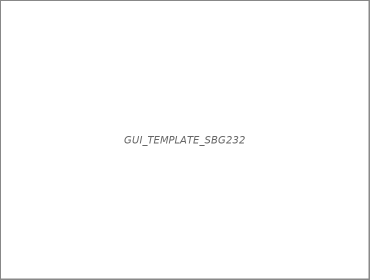
VISUALIZATION GUI_SBG232_SIM  // 370x280
    Frame (0,0 370x280)
        shows GUI_TEMPLATE_SBG232(m_Instance := MAIN.sbg232_sim)
END_VISUALIZATION

(* stored: Version 1.1.0.1, ProductVersion 3.1.4024.12
   Visu GUI_SBG232_SIM: Id {af8018f8-06c7-4b23-aad0-1f1dba0308bd} *)
